{attribute 'GeneratedUsingTerminal: EL3681-0000-0017'}
{attribute addProperty BoxType "EL3681-0000-0017"}
{attribute addProperty Id "StatusAT %I*Status_237FCB0F10ValueAT %I*DINT4"}
{attribute addProperty CRC "981700113"}
{attribute addProperty Size "14"}
TYPE SAI_Inputs_3A838E11 EXTENDS InputBase_8311D824 :
STRUCT
	{attribute addProperty Name "Status"}
	Status AT %I* : Status_237FCB0F;
	{attribute addProperty Name "Value"}
	Value AT %I* : DINT;
END_STRUCT
END_TYPE

(* stored: Version 1.2.0.0, ProductVersion 3.1.4024.9
   DUT SAI_Inputs_3A838E11: Id {567fb342-c4f2-4943-a88a-8281ebd5a22e} *)
